// TIA Portal V17 export
// export: Created 2025-06-26T07:49:58.1035314Z, ExportSetting WithDefaults, DisplayName Totally Integrated Automation Portal, DisplayVersion V17 Update 8, DisplayName TIA Portal Openness, DisplayVersion V17 Update 8, DisplayName TIA Portal Version Control Interface, DisplayVersion V17, DisplayName STEP 7 Professional, DisplayVersion V17 Update 8, DisplayName STEP 7 Safety, DisplayVersion V17 Update 6, DisplayName WinCC Advanced, DisplayVersion V17 Update 8
TYPE "VariableSetting-STRUCT"
// stored: IsFailsafeCompliant false
   STRUCT
      SystemType : Int;   // Select the used system type
      CompressorType : Int;   // Select the used compressor type
      FluidType : Int;   // Select the used working fluid
      OilPreheating_acv : Bool;   // Activates the oil heaters for pre-heating in state standby
      OilHeatSetpoint_min : Real := 10.0;   // Lowest possible oil heater temperature setpoint
      EnableViaHMI : Bool;   // Allow HMI to start & stop the HB
      EnableViaApplication : Bool;   // Allow the Application PLC to start & stop the HB
      SourceOkFromApplication : Bool;
      SinkOkFromApplication : Bool;
      HeatSourceExternalControl : Bool;   // Heat source auxiliary equipment controlled externally
      HeatSinkExternalControl : Bool;   // Heat sink auxiliary equipment controlled externally
   END_STRUCT;
END_TYPE
